{attribute 'qualified_only'}
{attribute 'strict'}
TYPE EStampStates :
(
	none := 0,
	unpressed := 1,
	pressed := 2,
	busy := 3
) UINT;
END_TYPE

(* stored: Version 1.1.0.1
   DUT EStampStates: Id {afeb4440-48f0-48ae-821b-e0952fe1a770} *)
